			bReadDecPointVehicle := FALSE;	// Done in M_StateMachineNode_ADS
			bReadDecPointVehicleBusy := TRUE;
			bReturn := TRUE;			
		ELSE
	// NEW!!!
			// NOTE: iReadIndex is MagneMotion vehicle No
			REPEAT
				iReadIndex := iReadIndex + 1;
				IF (M_CheckVehicleOwned(iReadIndex)) THEN
					// Vehicle is owned by this cell... Read data from Track Server for this vehicle
					IF (M_CheckVehicleEventRead(iReadIndex)) THEN
						// Vehicle data is selected to be read! (event-based reading)
						EXIT;
					END_IF
				ELSIF (M_CheckVehicleSurvail(iReadIndex)) THEN
					// Vehicle is survailed by this cell (read data continously!)... Read data from Track Server for this vehicle
					EXIT;
				ELSIF (iReadIndex <> nDecisionPointVehicleNo) THEN
					// Not owned or surveilled or being handled by decision point. Delete any previous read data
					IF (iReadIndex > 0 AND iReadIndex <= MM_MAX_NUMBER_OF_VEHICLE_ELEMENTS) THEN
						aReadVehicleData[iReadIndex].stVehicle.bDataValid := FALSE;
					END_IF
				END_IF
				UNTIL (iReadIndex >= MM_MAX_NUMBER_OF_VEHICLE_ELEMENTS)
			END_REPEAT
			
			IF (iReadIndex <= MM_MAX_NUMBER_OF_VEHICLE_ELEMENTS) THEN
				// Build remote symbol name
				sPrefix := CONCAT(sObjectIDentifier, '.stTrackStatus');
				// Data pointer for received data
				pReadNodeData := ADR(aReadVehicleData[iReadIndex].stVehicle);
				// Header data size
				cbDataTotal := SIZEOF(aReadVehicleData[iReadIndex].stVehicle);
				
				// Specify nodes to read by variable name
				sTrackServerSymbol := CONCAT(sPrefix, '.aVehicles[');
				sTrackServerSymbol := CONCAT(sTrackServerSymbol, UINT_TO_STRING(iReadIndex));
				sTrackServerSymbol := CONCAT(sTrackServerSymbol, ']');
				
				// Remove this vehicle from the event-driven reading list
				M_VehicleToReadRemove(iReadIndex);
				
				bReturn := TRUE;
			ELSE
				// Read next type
				iReadIndex := 0;
				eReadType := E_OPC_NodeType.Paths;
				bReturn := FALSE;
			END_IF
	// NEW END!!!	
			// Select vehicle to read data from (only the vehicles this cell is responsible for)
(*			REPEAT
				iReadIndex := iReadIndex+1;
				IF (iReadIndex > MM_MAX_NUMBER_OF_VEHICLE_ELEMENTS) THEN
					EXIT;
				END_IF
				UNTIL (aReadCellData.stCell.anVehicles[iReadIndex] > 0)
			END_REPEAT
			IF (iReadIndex <= MM_MAX_NUMBER_OF_VEHICLE_ELEMENTS) THEN
				// Build remote symbol name
				sPrefix := CONCAT(sObjectIDentifier, '.stTrackStatus');
				// Data pointer for received data
				pReadNodeData := ADR(aReadVehicleData[aReadCellData.stCell.anVehicles[iReadIndex]].stVehicle);
				// Header data size
				cbDataTotal := SIZEOF(aReadVehicleData[aReadCellData.stCell.anVehicles[iReadIndex]].stVehicle);
				
				// Specify nodes to read by variable name
				sTrackServerSymbol := CONCAT(sPrefix, '.aVehicles[');
				sTrackServerSymbol := CONCAT(sTrackServerSymbol, UINT_TO_STRING(aReadCellData.stCell.anVehicles[iReadIndex]));
				sTrackServerSymbol := CONCAT(sTrackServerSymbol, ']');
				bReturn := TRUE;
			ELSE
				// Read next type
				iReadIndex := 0;
				eReadType := E_OPC_NodeType.Paths;
				bReturn := FALSE;
			END_IF		*)
		END_IF
		
	E_OPC_NodeType.Paths:
		// Select path to read data from
		REPEAT
			iReadIndex := iReadIndex+1;
			IF (iReadIndex > MM_MAX_NUMBER_OF_PATH_ELEMENTS) THEN
				EXIT;
			END_IF
			UNTIL (abControlledPaths[iReadIndex])
		END_REPEAT
		IF ((iReadIndex <= MM_MAX_NUMBER_OF_PATH_ELEMENTS) AND NOT tonSkipPathRead.Q) THEN	// Skip path reading when paths are started!
			// Build remote symbol name
			sPrefix := CONCAT(sObjectIDentifier, '.stTrackStatus');
			// Data pointer for received data
			pReadNodeData := ADR(aReadPathData[iReadIndex].stPathData);
			// Header data size
			cbDataTotal := SIZEOF(aReadPathData[iReadIndex].stPathData);
			
			// Specify nodes to read by variable name
			sTrackServerSymbol := CONCAT(sPrefix, '.aPaths[');
			sTrackServerSymbol := CONCAT(sTrackServerSymbol, UINT_TO_STRING(iReadIndex));
			sTrackServerSymbol := CONCAT(sTrackServerSymbol, ']');
			bReturn := TRUE;
		ELSE
			// Read next type
			iReadIndex := 0;
			eReadType := E_OPC_NodeType.Stations;
			bReturn := FALSE;
		END_IF
		
	E_OPC_NodeType.Stations:
		// Select Station to read data from
// TEST
		IF (M_CheckStationsRead()) THEN
			// Index for station data from track server has been found... Only read these stations
			REPEAT
				iReadIndex := iReadIndex+1;
				IF (iReadIndex > MM_MAX_NUMBER_OF_STATION_ELEMENTS) THEN
					EXIT;
				END_IF
				UNTIL (M_CheckStationIndex(iReadIndex))
			END_REPEAT
		ELSE
			// Index for station data from track server has NOT been found... Read data from all stations
			iReadIndex := iReadIndex + 1;
		END_IF
// TEST END
//		iReadIndex := iReadIndex+1;
		IF (iReadIndex <= MM_MAX_NUMBER_OF_STATION_ELEMENTS) THEN
			// Build remote symbol name
			sPrefix := CONCAT(sObjectIDentifier, '.stTrackStatus');
			// Data pointer
			pReadNodeData := ADR(aReadStationData[iReadIndex].stStationData);
			// Header data
			cbDataTotal := SIZEOF(aReadStationData[iReadIndex].stStationData);
			
			// Specify nodes to read by variable name
			sTrackServerSymbol := CONCAT(sPrefix, '.aStations[');
			sTrackServerSymbol := CONCAT(sTrackServerSymbol, UINT_TO_STRING(iReadIndex));
			sTrackServerSymbol := CONCAT(sTrackServerSymbol, ']');
			bReturn := TRUE;
		ELSE
			// Read next type
			iReadIndex := 0;
			eReadType := E_OPC_NodeType.Cells;
			bReturn := FALSE;
		END_IF
	
	E_OPC_NodeType.Cells:
		// Select Station to read data from
		iReadIndex := iThisCellIndex;
		IF (iReadIndex > 0 AND iReadIndex <= MM_MAX_NUMBER_OF_CELL_ELEMENTS) THEN
			// Build remote symbol name
			sPrefix := CONCAT(sObjectIDentifier, '.stTrackStatus');
			// Data pointer
			pReadNodeData := ADR(aReadCellData.stCell);
			// Header data
			cbDataTotal := SIZEOF(aReadCellData.stCell);
			
			// Specify nodes to read by variable name
			sTrackServerSymbol := CONCAT(sPrefix, '.aCells[');
			sTrackServerSymbol := CONCAT(sTrackServerSymbol, UINT_TO_STRING(iReadIndex));
			sTrackServerSymbol := CONCAT(sTrackServerSymbol, ']');
			bReturn := TRUE;

			// continue to next type after this read!
			iReadIndex := 0;
			bReadDecPointVehicle := TRUE;	// Force reading of the vehicle at decision point before other vehicles
			IF (NOT bReadDecPointCellDone) THEN
				bReadDecPointCell := TRUE;
			END_IF
			eReadType := E_OPC_NodeType.Vehicles;
		ELSE
			// Read next type
			iReadIndex := 0;
			bReadDecPointVehicle := TRUE;	// Force reading of the vehicle at decision point before other vehicles
			eReadType := E_OPC_NodeType.Vehicles;
			bReturn := FALSE;
		END_IF

END_CASE

M_InitNodeData_ADS := bReturn;
END_METHOD

METHOD PROTECTED M_InitNodeData_OPCUA : BOOL
VAR
	i		: UINT;
	sPrefix : STRING;
END_VAR
VAR
	cbDataTotal2 : UINT;
END_VAR
// NOTE!!!
// Maximum of 10 elements to read for each Node List reading!


(* Node data, init to use string identifier and set namespace index *)
FOR i:=1 TO nMaxNodeIDsInList BY 1 DO
	aNodeIDs[i].eIdentifierType := eUAIdentifierType_String;
	aNodeIDs[i].nNamespaceIndex := nNameSpaceIndexNodes;
END_FOR

nNoOfNodes := 0;
cbDataTotal := 0;

// TEST
eReadType := E_OPC_NodeType.Nodes;
iReadIndex := 1;

// Comm type selection
CASE eReadType OF
	E_OPC_NodeType.Vehicles:
		// Limit number of elements
		iReadIndex := LIMIT(1, iReadIndex, MM_MAX_NUMBER_OF_VEHICLE_ELEMENTS);
		// Build remote symbol name
		sPrefix := CONCAT(sObjectIDentifier, '.stTrackStatus.aVehicles[');
		sPrefix := CONCAT(sPrefix, UINT_TO_STRING(iReadIndex));
		sPrefix := CONCAT(sPrefix, ']');
		// Data pointer
		pReadNodeData := ADR(aReadVehicleData[iReadIndex]);
		// Header data
		cbDataTotal := SIZEOF(aReadVehicleData[iReadIndex].stReadListReturnInfo);
		
		// Specify nodes to read by variable name
		nNoOfNodes := nNoOfNodes + 1;
		aNodeIDs[nNoOfNodes].sIdentifier := CONCAT(sPrefix, '.nVehicleID');
		acbDatas[nNoOfNodes] := SIZEOF(aReadVehicleData[iReadIndex].nVehicleID);
		cbDataTotal := cbDataTotal + acbDatas[nNoOfNodes];
		
		nNoOfNodes := nNoOfNodes + 1;
		aNodeIDs[nNoOfNodes].sIdentifier := CONCAT(sPrefix, '.bVehiclePresent');
		acbDatas[nNoOfNodes] := SIZEOF(aReadVehicleData[iReadIndex].bVehiclePresent);
		cbDataTotal := cbDataTotal + acbDatas[nNoOfNodes];
		
		nNoOfNodes := nNoOfNodes + 1;
		aNodeIDs[nNoOfNodes].sIdentifier := CONCAT(sPrefix, '.nState');
		acbDatas[nNoOfNodes] := SIZEOF(aReadVehicleData[iReadIndex].nState);
		cbDataTotal := cbDataTotal + acbDatas[nNoOfNodes];
		
		nNoOfNodes := nNoOfNodes + 1;
		aNodeIDs[nNoOfNodes].sIdentifier := CONCAT(sPrefix, '.nPathID');
		acbDatas[nNoOfNodes] := SIZEOF(aReadVehicleData[iReadIndex].nPathID);
		cbDataTotal := cbDataTotal + acbDatas[nNoOfNodes];
		
		nNoOfNodes := nNoOfNodes + 1;
		aNodeIDs[nNoOfNodes].sIdentifier := CONCAT(sPrefix, '.fPosition');
		acbDatas[nNoOfNodes] := SIZEOF(aReadVehicleData[iReadIndex].fPosition);
		cbDataTotal := cbDataTotal + acbDatas[nNoOfNodes];
		
		nNoOfNodes := nNoOfNodes + 1;
		aNodeIDs[nNoOfNodes].sIdentifier := CONCAT(sPrefix, '.nTargetPathID');
		acbDatas[nNoOfNodes] := SIZEOF(aReadVehicleData[iReadIndex].nTargetPathID);
		cbDataTotal := cbDataTotal + acbDatas[nNoOfNodes];
		
		nNoOfNodes := nNoOfNodes + 1;
		aNodeIDs[nNoOfNodes].sIdentifier := CONCAT(sPrefix, '.fTargetPosition');
		acbDatas[nNoOfNodes] := SIZEOF(aReadVehicleData[iReadIndex].fTargetPosition);
		cbDataTotal := cbDataTotal + acbDatas[nNoOfNodes];
		
		nNoOfNodes := nNoOfNodes + 1;
		aNodeIDs[nNoOfNodes].sIdentifier := CONCAT(sPrefix, '.fVelocity');
		acbDatas[nNoOfNodes] := SIZEOF(aReadVehicleData[iReadIndex].fVelocity);
		cbDataTotal := cbDataTotal + acbDatas[nNoOfNodes];
				
		// Read next vehicle value
		iReadIndex := iReadIndex+1;;
		IF (iReadIndex > MM_MAX_NUMBER_OF_VEHICLE_ELEMENTS) THEN
			// Read next type
			iReadIndex := 0;
			eReadType := E_OPC_NodeType.Paths;
		END_IF

	E_OPC_NodeType.Paths:
		// Limit number of elements
		iReadIndex := LIMIT(1, iReadIndex, MM_MAX_NUMBER_OF_PATH_ELEMENTS);
		// Build remote symbol name
		sPrefix := CONCAT(sObjectIDentifier, '.stTrackStatus.aPaths[');
		sPrefix := CONCAT(sPrefix, UINT_TO_STRING(iReadIndex));
		sPrefix := CONCAT(sPrefix, ']');
		// Data pointer
		pReadNodeData := ADR(aReadPathData[iReadIndex]);
		
		// Header data
		cbDataTotal := SIZEOF(aReadPathData[iReadIndex].stReadListReturnInfo);
		
		// Specify nodes to read by variable name
		nNoOfNodes := nNoOfNodes + 1;
		aNodeIDs[nNoOfNodes].sIdentifier := CONCAT(sPrefix, '.nPathID');
		acbDatas[nNoOfNodes] := SIZEOF(aReadPathData[iReadIndex].nPathID);
		cbDataTotal := cbDataTotal + acbDatas[nNoOfNodes];

		nNoOfNodes := nNoOfNodes + 1;
		aNodeIDs[nNoOfNodes].sIdentifier := CONCAT(sPrefix, '.sCellID');
		acbDatas[nNoOfNodes] := SIZEOF(aReadPathData[iReadIndex].sCellID);
		cbDataTotal := cbDataTotal + acbDatas[nNoOfNodes];

		nNoOfNodes := nNoOfNodes + 1;
		aNodeIDs[nNoOfNodes].sIdentifier := CONCAT(sPrefix, '.bPathPresent');
		acbDatas[nNoOfNodes] := SIZEOF(aReadPathData[iReadIndex].bPathPresent);
		cbDataTotal := cbDataTotal + acbDatas[nNoOfNodes];

		nNoOfNodes := nNoOfNodes + 1;
		aNodeIDs[nNoOfNodes].sIdentifier := CONCAT(sPrefix, '.nState');
		acbDatas[nNoOfNodes] := SIZEOF(aReadPathData[iReadIndex].nState);
		cbDataTotal := cbDataTotal + acbDatas[nNoOfNodes];

		// Read next path value
		iReadIndex := iReadIndex+1;
		IF (iReadIndex > MM_MAX_NUMBER_OF_PATH_ELEMENTS) THEN
			// Read next type
			iReadIndex := 0;
			eReadType := E_OPC_NodeType.Nodes;
			//eReadType := E_OPC_NodeType.Vehicles;
		END_IF
		
		
	E_OPC_NodeType.Nodes:
		// Limit number of elements
		iReadIndex := LIMIT(1, iReadIndex, 10);
		// Build remote symbol name
		sPrefix := CONCAT(sObjectIDentifier, '.stTrackStatus');
		// Data pointer
		pReadNodeData := ADR(aReadNodeData[iReadIndex]);
		
		// Header data
		cbDataTotal := SIZEOF(aReadNodeData[iReadIndex].stReadListReturnInfo);
		cbDataTotal2 := SIZEOF(aReadNodeData[iReadIndex]);
		
		// Specify nodes to read by variable name
		nNoOfNodes := nNoOfNodes + 1;
		aNodeIDs[nNoOfNodes].sIdentifier := CONCAT(sPrefix, '.aNodes[');
		aNodeIDs[nNoOfNodes].sIdentifier := CONCAT(aNodeIDs[nNoOfNodes].sIdentifier, UINT_TO_STRING(iReadIndex));
		aNodeIDs[nNoOfNodes].sIdentifier := CONCAT(aNodeIDs[nNoOfNodes].sIdentifier, ']');
		acbDatas[nNoOfNodes] := SIZEOF(aReadNodeData[iReadIndex].stNodeData);
		cbDataTotal := cbDataTotal + acbDatas[nNoOfNodes];

		// Read next node value
		iReadIndex := iReadIndex+1;
		IF (iReadIndex > 10) THEN
			// Read next type
			iReadIndex := 0;
			eReadType := E_OPC_NodeType.Vehicles;
		END_IF

END_CASE
END_METHOD

METHOD PROTECTED M_MappingData
VAR_INPUT
END_VAR
VAR
	i			: USINT;
	iRes		: UINT;
END_VAR
// Handle the mapping data from OPC UA (stCommand)

CASE eMappingDataState OF
	// Init state
	E_MappingDataState.Undefined:
		eMappingDataState := E_MappingDataState.CheckRequest;
	
	// Check command data request
	E_MappingDataState.CheckRequest:
		IF ((stMappingIn.ChangeRequest <> stMappingOut.ChangeStatus) AND (stMappingIn.ChangeRequest > 0)) THEN
			// Check if changes is allowed on mapping data (from LC)
			IF (stAdditionalDataIn.MESHandShakes.DataChangeStatusTransportMapping = stMappingOut.DataChange) THEN
				stMappingOut.ChangeAcknowlegde := stMappingIn.ChangeRequest;
				stMappingOut.DataChange := stMappingOut.DataChange + 1;
				
				// Find vehicle ID with specified carrier ID
				iMappingDataVehicleID := M_CarrierIDToVehicleID(stMappingIn.Carrier.CarrierID);
	
				// Check vehicle number
				IF (iMappingDataVehicleID > 0) THEN
					eMappingDataState := E_MappingDataState.UpdateMappingData;
				ELSE
					eMappingDataState := E_MappingDataState.Error;
				END_IF
			END_IF	
		END_IF	
	
	// Perform data update
	E_MappingDataState.UpdateMappingData:
		iRes := M_CallUpdateVehicleMappingData(	nVehicleID := iMappingDataVehicleID,
												sCarrierID := stMappingIn.Carrier.CarrierID, 
												bTool := stMappingIn.Carrier.Tool, 
												sToolID := stMappingIn.Carrier.ToolID, 
												bMaterial := stMappingIn.Carrier.Material,
												sMaterialID := stMappingIn.Carrier.MaterialID 	);
		IF (iRes = 2) THEN
			// Success.
			eMappingDataState := E_MappingDataState.UpdateReworkData;
		ELSIF (iRes = 3) THEN
			// Error!
			eMappingDataState := E_MappingDataState.Error;
		END_IF
	
	// Perform rework update
	E_MappingDataState.UpdateReworkData:
		iRes := M_CallUpdateVehicleReworkData(	nVehicleID := iMappingDataVehicleID,
												sCarrierID := stMappingIn.Carrier.CarrierID,
												bNOK := stMappingIn.Carrier.NOK	); 
		IF (iRes = 2) THEN
			// Success..
			eMappingDataState := E_MappingDataState.Done;
		ELSIF (iRes = 3) THEN
			// Error!
			eMappingDataState := E_MappingDataState.Error;
		END_IF
	
	E_MappingDataState.Done:
		// Completed... Update output mapping data
		stMappingOut.ValidRequest := TRUE;
		stMappingOut.Carrier := stMappingIn.Carrier;
		stMappingOut.StationBuffer := stMappingIn.StationBuffer;
		stMappingOut.ChangeStatus := stMappingIn.ChangeRequest;
		stMappingOut.DataChange := stMappingOut.DataChange + 1;
		eMappingDataState := E_MappingDataState.Undefined;
	
	E_MappingDataState.Error:
		// Error... Valid request = FALSE
		stMappingOut.ValidRequest := FALSE;
		stMappingOut.ChangeStatus := stMappingIn.ChangeRequest;
		stMappingOut.DataChange := stMappingOut.DataChange + 1;
		eMappingDataState := E_MappingDataState.Undefined;
	
END_CASE
END_METHOD

METHOD PROTECTED M_ReworkData
VAR_INPUT
END_VAR
VAR
	i			: USINT;
	iRes		: UINT;
END_VAR
// Handle the mapping data from OPC UA (stCommand)

CASE eReworkDataState OF
	// Init state
	E_ReworkDataState.Undefined:
		bReworkValue := FALSE;
		iReworkDataStation := 0;
		iReworkDataStationNo := 0;
		eReworkDataState := E_ReworkDataState.CheckRequest;
	
	// Check command data request
	E_ReworkDataState.CheckRequest:
		FOR i := 1 TO 5 BY 1 DO
			/////////////////////////////////////////////////////////////////////////////////////////////////////////////////////
			// Rework completed from station (shoe rework is done handled)
			/////////////////////////////////////////////////////////////////////////////////////////////////////////////////////
			IF (abStation1ReworkDone[i]) THEN
				iReworkDataStation := i;
				iReworkDataStationNo := 1;

				// Check vehicle at station
				iReworkDataVehicleID := aStations[iReworkDataStation].stStationData1.nCurrentVehicleID;
				IF ((iReworkDataVehicleID > 0) AND (iReworkDataVehicleID <= MM_MAX_NUMBER_OF_VEHICLE_ELEMENTS) ) THEN
					// There is a vehicle on that station! Get the Carrier ID
					sReworkDataCarrierID := aReadVehicleData[iReworkDataVehicleID].stVehicle.sCarrierID;
					
					// Check carrier ID of vehicle
					IF (sReworkDataCarrierID <> '') THEN
						bReworkValue := FALSE;	// Set carrier status to rework NOT needed!
						eReworkDataState := E_ReworkDataState.UpdateReworkData;
					ELSE
						// Error!
						eReworkDataState := E_ReworkDataState.Error;
					
					END_IF
				ELSE
					// Error!
					eReworkDataState := E_ReworkDataState.Error;
				
				END_IF

				EXIT;
				
			ELSIF (abStation2ReworkDone[i]) THEN
				iReworkDataStation := i;
				iReworkDataStationNo := 2;

				iReworkDataVehicleID := aStations[iReworkDataStation].stStationData2.nCurrentVehicleID;
				IF ((iReworkDataVehicleID > 0) AND (iReworkDataVehicleID <= MM_MAX_NUMBER_OF_VEHICLE_ELEMENTS) ) THEN
					// There is a vehicle on that station! Get the Carrier ID
					sReworkDataCarrierID := aReadVehicleData[iReworkDataVehicleID].stVehicle.sCarrierID;
					
					// Check carrier ID of vehicle
					IF (sReworkDataCarrierID <> '') THEN
						bReworkValue := FALSE;	// Set carrier status to rework NOT needed!
						eReworkDataState := E_ReworkDataState.UpdateReworkData;
					ELSE
						// Error!
						eReworkDataState := E_ReworkDataState.Error;
					
					END_IF				
				ELSE
					// Error!
					eReworkDataState := E_ReworkDataState.Error;
				
				END_IF

				EXIT;

			/////////////////////////////////////////////////////////////////////////////////////////////////////////////////////
			// Rework request from station (shoe needs to be reworked)
			/////////////////////////////////////////////////////////////////////////////////////////////////////////////////////
			ELSIF (abStation1ReworkReq[i]) THEN
				iReworkDataStation := i;
				iReworkDataStationNo := 1;

				// Check vehicle at station
				iReworkDataVehicleID := aStations[iReworkDataStation].stStationData1.nCurrentVehicleID;
				IF ((iReworkDataVehicleID > 0) AND (iReworkDataVehicleID <= MM_MAX_NUMBER_OF_VEHICLE_ELEMENTS) ) THEN
					// There is a vehicle on that station! Get the Carrier ID
					sReworkDataCarrierID := aReadVehicleData[iReworkDataVehicleID].stVehicle.sCarrierID;
					
					// Check carrier ID of vehicle
					IF (sReworkDataCarrierID <> '') THEN
						bReworkValue := TRUE;	// Set carrier status to rework needed!
						eReworkDataState := E_ReworkDataState.UpdateReworkData;
					ELSE
						// Error!
						eReworkDataState := E_ReworkDataState.Error;
					
					END_IF
				ELSE
					// Error!
					eReworkDataState := E_ReworkDataState.Error;
				
				END_IF

				EXIT;
				
			ELSIF (abStation2ReworkReq[i]) THEN
				iReworkDataStation := i;
				iReworkDataStationNo := 2;

				iReworkDataVehicleID := aStations[iReworkDataStation].stStationData2.nCurrentVehicleID;
				IF ((iReworkDataVehicleID > 0) AND (iReworkDataVehicleID <= MM_MAX_NUMBER_OF_VEHICLE_ELEMENTS) ) THEN
					// There is a vehicle on that station! Get the Carrier ID
					sReworkDataCarrierID := aReadVehicleData[iReworkDataVehicleID].stVehicle.sCarrierID;
					
					// Check carrier ID of vehicle
					IF (sReworkDataCarrierID <> '') THEN
						bReworkValue := TRUE;	// Set carrier status to rework needed!
						eReworkDataState := E_ReworkDataState.UpdateReworkData;
					ELSE
						// Error!
						eReworkDataState := E_ReworkDataState.Error;
					
					END_IF				
				ELSE
					// Error!
					eReworkDataState := E_ReworkDataState.Error;
				
				END_IF

				EXIT;
			END_IF
		END_FOR
	
	// Perform rework update
	E_ReworkDataState.UpdateReworkData:
		iRes := M_CallUpdateVehicleReworkData(	nVehicleID := iReworkDataVehicleID,
												sCarrierID := sReworkDataCarrierID,
												bNOK := bReworkValue 	);
		IF (iRes = 2) THEN
			// Success..
			F_LogLine(CONCAT('TC_RWK: Vehicle ', CONCAT(UINT_TO_STRING(iReworkDataVehicleID), ' NOK set to %d')), BOOL_TO_DINT(bReworkValue));
			eReworkDataState := E_ReworkDataState.Done;
		ELSIF (iRes = 3) THEN
			// Error!
			eReworkDataState := E_ReworkDataState.Error;
		END_IF
	
	E_ReworkDataState.Done:
		// Completed... Wait until activation bit is sert to FALSE (when vehicle has been removed from station)
		IF (bReworkValue) THEN
			IF (iReworkDataStationNo = 1) THEN
				IF (NOT abStation1ReworkReq[iReworkDataStation]) THEN
					eReworkDataState := E_ReworkDataState.Undefined;		
				END_IF
	
			ELSIF (iReworkDataStationNo = 2) THEN
				IF (NOT abStation2ReworkReq[iReworkDataStation]) THEN
					eReworkDataState := E_ReworkDataState.Undefined;
				END_IF
	
			END_IF
		ELSE
			IF (iReworkDataStationNo = 1) THEN
				IF (NOT abStation1ReworkDone[iReworkDataStation]) THEN
					eReworkDataState := E_ReworkDataState.Undefined;		
				END_IF
	
			ELSIF (iReworkDataStationNo = 2) THEN
				IF (NOT abStation2ReworkDone[iReworkDataStation]) THEN
					eReworkDataState := E_ReworkDataState.Undefined;
				END_IF
	
			END_IF
		END_IF
	
	E_ReworkDataState.Error:
		// Error... Wait until activation bit is sert to FALSE (when vehicle has been removed from station)
		// TODO!!! Alarm!
		IF (bReworkValue) THEN
			IF (iReworkDataStationNo = 1) THEN
				IF (NOT abStation1ReworkReq[iReworkDataStation]) THEN
					eReworkDataState := E_ReworkDataState.Undefined;		
				END_IF
	
			ELSIF (iReworkDataStationNo = 2) THEN
				IF (NOT abStation2ReworkReq[iReworkDataStation]) THEN
					eReworkDataState := E_ReworkDataState.Undefined;
				END_IF
	
			END_IF
		ELSE
			IF (iReworkDataStationNo = 1) THEN
				IF (NOT abStation1ReworkDone[iReworkDataStation]) THEN
					eReworkDataState := E_ReworkDataState.Undefined;		
				END_IF
	
			ELSIF (iReworkDataStationNo = 2) THEN
				IF (NOT abStation2ReworkDone[iReworkDataStation]) THEN
					eReworkDataState := E_ReworkDataState.Undefined;
				END_IF
	
			END_IF
		END_IF

END_CASE
END_METHOD

METHOD PROTECTED M_Run : BOOL
VAR_INPUT
END_VAR
VAR
	i	: USINT;
END_VAR
// Get system time
fbGetTime(	NETID:= '',	// Local PLC 
			START:= NOT fbGetTime.START AND NOT fbGetTime.BUSY, 
			TMOUT:= T#5S	);

///////////////////////////////////////////////////////////////////////////////////////////////////////////////////
// FB's for method calling
///////////////////////////////////////////////////////////////////////////////////////////////////////////////////
	(* Handle server connect *)
	fbConnectMethod(	Execute				:= , 
						ServerUrl			:= sTrackServerUrl, 
						SessionConnectInfo	:= stConnectInfoMethod, 
						Timeout				:= T#10S, 
						ConnectionHdl		=> , 
						Done				=> , 
						Busy				=> , 
						Error				=> , 
						ErrorID				=> 	);
					
	(* Handle server dicconnect *)
	fbDisconnectMethod(	Execute				:= , 
						ConnectionHdl		:= nConnectHdlMethod, 
						Timeout				:= T#10S, 
						Done				=> , 
						Busy				=> , 
						Error				=> , 
						ErrorID				=> 	);
						
	(* Get namepsace *)
	fbGetNamespaceMethod(	Execute				:= , 
							ConnectionHdl		:= nConnectHdlMethod, 
							NamespaceUri		:= sNameSpaceUri, 
							Timeout				:= T#10S, 
							NamespaceIndex		=> , 
							Done				=> , 
							Busy				=> , 
							Error				=> , 
							ErrorID				=> 	);
	
	(* Get method handle *)
	stObjectNodeID.nNamespaceIndex := nNameSpaceIndexMethod;
	stObjectNodeID.sIdentifier := sObjectIDentifier;
	stMethodNodeID.nNamespaceIndex := nNameSpaceIndexMethod;
	stMethodNodeID.sIdentifier := sMethodIdentifier;
	fbGetHandleMethod(	Execute				:= , 
						ConnectionHdl		:= nConnectHdlMethod, 
						ObjectNodeID		:= stObjectNodeID, 
						MethodNodeID		:= stMethodNodeID, 
						Timeout				:= T#10S, 
						MethodHdl			=> , 
						Done				=> , 
						Busy				=> , 
						Error				=> , 
						ErrorID				=>	);
	
	(* Call method *)
	fbCallMethod(	Execute					:= , 
					ConnectionHdl			:= nConnectHdlMethod, 
					MethodHdl				:= nHandleMethod, 
					nNumberOfInputArguments	:= , 
					pInputArgInfo			:= , 
					cbInputArgInfo			:= , 
					pInputArgData			:= , 
					cbInputArgData			:= , 
					pInputWriteData			:= 0,
					cbInputWriteData		:= 0,
					nNumberOfOutputArguments:= , 
					pOutputArgInfo			:= , 
					cbOutputArgInfo			:= , 
					pOutputArgInfoAndData	:= , 
					cbOutputArgInfoAndData	:= , 
					Timeout					:= T#10S, 
					cbRead_R				=> , 
					Done					=> , 
					Busy					=> , 
					Error					=> , 
					ErrorID					=> );
	
	(* Release method handle *)
	fbReleaseHandleMethod(	Execute			:= , 
							ConnectionHdl	:= nConnectHdlMethod, 
							MethodHdl		:= nHandleMethod, 
							Timeout			:= T#10S, 
							Done			=> , 
							Busy			=> , 
							Error			=> , 
							ErrorID			=> 	);

///////////////////////////////////////////////////////////////////////////////////////////////////////////////////
// FB's for method calling
///////////////////////////////////////////////////////////////////////////////////////////////////////////////////
	(* Handle server connect *)
	fbConnectNodes(	Execute				:= , 
					ServerUrl			:= sTrackServerUrl, 
					SessionConnectInfo	:= stConnectInfoNodes, 
					Timeout				:= T#10S, 
					ConnectionHdl		=> , 
					Done				=> , 
					Busy				=> , 
					Error				=> , 
					ErrorID				=> 	);
					
	(* Handle server dicconnect *)
	fbDisconnectNodes(	Execute				:= , 
						ConnectionHdl		:= nConnectHandleNodes, 
						Timeout				:= T#10S, 
						Done				=> , 
						Busy				=> , 
						Error				=> , 
						ErrorID				=> 	);
						
	(* Get namepsace *)
	fbGetNamespaceNodes(	Execute				:= , 
						ConnectionHdl		:= nConnectHandleNodes, 
						NamespaceUri		:= sNameSpaceUri, 
						Timeout				:= T#10S, 
						NamespaceIndex		=> , 
						Done				=> , 
						Busy				=> , 
						Error				=> , 
						ErrorID				=> 	);
	
	(* Get node handle *)
	fbGetHandleNodes(	Execute				:= , 
						ConnectionHdl		:= nConnectHandleNodes, 
						NodeIDCount			:= nNoOfNodes,
						NodeIDs				:= aNodeIDs, 
						Timeout				:= T#10S, 
						NodeHdls			=> , 
						Done				=> , 
						Busy				=> , 
						Error				=> , 
						ErrorID				=> 	);
		
	(* Read node data *)
	fbReadNodes(	Execute:= , 
					ConnectionHdl			:= nConnectHandleNodes,
					NodeHdlCount			:= nNoOfNodes,
					NodeHdls				:= anHandleNodes, 
					stNodeAddInfo			:= astNodeAddInfo, 
					pVariable				:= pReadNodeData, 
					cbData					:= acbDatas,
					cbDataTotal				:= cbDataTotal, 
					Timeout					:= T#10S, 
					Done					=> , 
					Busy					=> , 
					Error					=> , 
					ErrorID					=> , 
					cbData_R				=> 	);
					
	(* Release node handle list *)
	fbReleaseHandleNodes(	Execute			:= , 
							ConnectionHdl	:= nConnectHandleNodes, 
							NodeHdlCount	:= nNoOfNodes, 
							NodeHdls		:= anHandleNodes, 
							Timeout			:= T#10S, 
							NodeErrorIDs	=> , 
							Done			=> , 
							Busy			=> , 
							Error			=> , 
							ErrorID			=> 	);
	
	(* Read interval *)
	tonReadInterval(	IN	:= ,
						PT	:= REAL_TO_TIME(rReadInterval * 1000.0),
						Q	=> ,
						ET	=> 	);
						
	(* Error automatic reset delay *)
	tonErrorReset(		IN	:= ,
						PT	:= REAL_TO_TIME(rErrorResetDelay * 1000.0),
						Q	=> ,
						ET	=> 	);

// Update Additional Data variables
	stAdditionaldataOut.bConnectedMethod := bConnectedMethod;
	stAdditionaldataOut.bConnectedNode := bConnectedNode;
	stAdditionaldataOut.bTrackReady := P_bTrackReady;
END_METHOD

METHOD PROTECTED M_StateMachine : BOOL
VAR_INPUT
END_VAR
VAR
	iRes	: INT;
	i		: UINT;
END_VAR

CASE eTrackState OF
	E_TrackState.Undefined:
		bStarted := FALSE;
		bSuspended := FALSE;
		iStationID := 1;
		iPathID := 1;
		iPathIndex := 1;
		IF (bConnectedMethod AND bConnectedNode) THEN
			// Communication connections established
			IF (bEnable) THEN
				eTrackState := E_TrackState.CheckInitDone;
			END_IF
		END_IF
	
	E_TrackState.CheckInitDone:
		// Check if track has been setup from this cell already on the track server
		iRes := M_CallGetCellIndex(sCellID);
		IF (iRes = 2) THEN
			// Success... Init done
			// Save found index
			iThisCellIndex := stGetCellIndexData.stOutput.nCellIndex;
			IF (iThisCellIndex > 0) THEN
				bTrackInitDone := TRUE;
				eTrackState := E_TrackState.Starting;
			ELSE
				bTrackInitDone := FALSE;
				bStationData1Done := FALSE;
				bStationData2Done := FALSE;
				// Clear station index
				FOR i := 1 TO 5 BY 1 DO
					iThisStationIndex[i] := 0;
				END_FOR
				eTrackState := E_TrackState.WaitAllowInit;
			END_IF
		ELSIF (iRes = 3) THEN
			// Error!
			// Clear station index
			FOR i := 1 TO 5 BY 1 DO
				iThisStationIndex[i] := 0;
			END_FOR
			eTrackState := E_TrackState.WaitAllowInit;
		END_IF
	
//	E_TrackState.InitDecisionPoint:
//		// Initialized with stations
//		eTrackState := E_TrackState.InitStations;
	
	E_TrackState.WaitAllowInit:
		// Initialized with stations
		IF (stAdditionalDataIn.bAllowInit) THEN
			stAdditionalDataIn.bAllowInit := FALSE;
			eTrackState := E_TrackState.InitStations;
		ELSIF (NOT bEnable OR NOT bConnectedMethod OR NOT bConnectedNode) THEN
			eTrackState := E_TrackState.Undefined;
		END_IF

	E_TrackState.InitStations:
		IF (aStations[iStationID].bPresent) THEN
			IF (aStations[iStationID].stStationData2.stLocation.nPathID > 0) THEN
				// Double position station
				iRes := M_CallAddStationDouble(nStationNo := iStationID);
				IF (iRes = 2) THEN
					// Success... Next station
					iStationID := iStationID + 1;
				ELSIF (iRes = 3) THEN
					// Error!
					// TODO!!!
					;				
				END_IF
			ELSE
				// Single position station
				iRes := M_CallAddStationSingle(nStationNo := iStationID);
				IF (iRes = 2) THEN
					// Success... Next station
					iStationID := iStationID + 1;
				ELSIF (iRes = 3) THEN
					// Error!
					// TODO!!!
					;				
				END_IF
			END_IF
		ELSE
			// Not enabled... Next station
			iStationID := iStationID + 1;
		END_IF
		IF (iStationID >= 5) THEN
			// All added
			iStationID := 1;
//			eTrackState := E_TrackState.InitPathsStations;	// init paths from stations, traffic lights and decision point 
			eTrackState := E_TrackState.SetPreBufferAdjust;
		END_IF
		
	E_TrackState.SetPreBufferAdjust:
		IF (aStations[iStationID].bPresent) THEN
			IF (aStationPreBufAdj[iStationID] <> 0.0) THEN
				iRes := M_CallAdjustBufferPosition(	nStationNo := iStationID,
													eBufferType := E_MMStationBuffer.eMMStationBuffer_PreProcess,
													rDistance := aStationPreBufAdj[iStationID]	);
				IF (iRes = 2) THEN
					// Success... Next station
					iStationID := iStationID + 1;
				ELSIF (iRes = 3) THEN
					// Error!
					// TODO!!!
					;
				END_IF
				
			ELSE
				// No adustment needed
				iStationID := iStationID + 1;
			END_IF
		ELSE
			// Not enabled... Next station
			iStationID := iStationID + 1;
		END_IF
		IF (iStationID >= 5) THEN
			// All checked/adjusted
			iStationID := 1;
			eTrackState := E_TrackState.SetPostBufferAdjust;
		END_IF
		
	E_TrackState.SetPostBufferAdjust:
		IF (aStations[iStationID].bPresent) THEN
			IF (aStationPostBufAdj[iStationID] <> 0.0) THEN
				iRes := M_CallAdjustBufferPosition(	nStationNo := iStationID,
													eBufferType := E_MMStationBuffer.eMMStationBuffer_PostProcess,
													rDistance := aStationPostBufAdj[iStationID]	);
				IF (iRes = 2) THEN
					// Success... Next station
					iStationID := iStationID + 1;
				ELSIF (iRes = 3) THEN
					// Error!
					// TODO!!!
					;
				END_IF
				
			ELSE
				// No adustment needed
				iStationID := iStationID + 1;
			END_IF
		ELSE
			// Not enabled... Next station
			iStationID := iStationID + 1;
		END_IF
		IF (iStationID >= 5) THEN
			// All checked/adjusted
			iStationID := 1;
			eTrackState := E_TrackState.InitPaths;
		END_IF
		
	// Create/init paths on track server for this cell
	E_TrackState.InitPaths:	
		IF (aPaths[iPathID] > 0) THEN
			iRes := M_CallAddPath(nPathNo := aPaths[iPathID]);
			IF (iRes = 2) THEN
				// Success... Next Path
				abControlledPaths[aPaths[iPathID]] := TRUE;
				iPathID := iPathID + 1;
			ELSIF (iRes = 3) THEN
				// Error!
				// TODO!!!
				;
			END_IF
		ELSE
			// All added
			iPathID := 1;
			eTrackState := E_TrackState.InitGetCellIndex;
		END_IF
(*		
	// Create/init paths on track server for this cell
	E_TrackState.InitPathsStations:	
		IF (aStations[iStationID].bPresent) THEN
			IF (NOT bStationData1Done) THEN
				iRes := M_CallAddPath(nPathNo := aStations[iStationID].stStationData1.stLocation.nPathID);
				IF (iRes = 2) THEN
					// Success... Next station
					abControlledPaths[aStations[iStationID].stStationData1.stLocation.nPathID] := TRUE;
					bStationData1Done := TRUE;
					IF (aStations[iStationID].stStationData1.stLocation.nPathID = aStations[iStationID].stStationData2.stLocation.nPathID) THEN
						// Station 2 is on the same path
						bStationData2Done := TRUE;
						iStationID := iStationID + 1;						
					ELSE
						// Station 2 is on a different path
						
					END_IF
				ELSIF (iRes = 3) THEN
					// Error!
					// TODO!!!
					;
				END_IF
			ELSIF (NOT bStationData2Done) THEN
				iRes := M_CallAddPath(nPathNo := aStations[iStationID].stStationData2.stLocation.nPathID);
				IF (iRes = 2) THEN
					// Success... Next station
					abControlledPaths[aStations[iStationID].stStationData2.stLocation.nPathID] := TRUE;
					bStationData2Done := TRUE;
					iStationID := iStationID + 1;
				ELSIF (iRes = 3) THEN
					// Error!
					// TODO!!!
					;
				END_IF
			END_IF
		ELSE
			// Not enabled... Next station
			iStationID := iStationID + 1;
		END_IF
		IF (iStationID >= 5) THEN
			// All added
			iStationID := 1;
			eTrackState := E_TrackState.InitPathsDecisionPoint;
		END_IF
	
	// Create/init paths on track server for this cell
	E_TrackState.InitPathsDecisionPoint:	
		IF (aStations[iStationID].bPresent) THEN
			iRes := M_CallAddPath(nPathNo := aStations[iStationID].stDecisionLocation.nPathID);
			IF (iRes = 2) THEN
				// Success... Next station
				abControlledPaths[aStations[iStationID].stDecisionLocation.nPathID] := TRUE;
				iStationID := iStationID + 1;
			ELSIF (iRes = 3) THEN
				// Error!
				// TODO!!!
				;
			END_IF
		ELSE
			// Not enabled... Next station
			iStationID := iStationID + 1;
		END_IF
		IF (iStationID >= 5) THEN
			// All added
			iStationID := 1;
			eTrackState := E_TrackState.InitPathsTrafficLight;
		END_IF

	// Create/init paths on track server for this cell
	E_TrackState.InitPathsTrafficLight:	
		IF (stTrafficLightLocation.nPathID > 0) THEN
			iRes := M_CallAddPath(nPathNo := stTrafficLightLocation.nPathID);	
			IF (iRes = 2) THEN
				// Success
				abControlledPaths[stTrafficLightLocation.nPathID] := TRUE;
				eTrackState := E_TrackState.InitGetCellIndex;
			ELSIF (iRes = 3) THEN
				// Error!
				// TODO!!!
				;
			END_IF
		ELSE
			eTrackState := E_TrackState.InitGetCellIndex;			
		END_IF
*)
	E_TrackState.InitGetCellIndex:
		iRes := M_CallGetCellIndex(sCellID);
		IF (iRes = 2) THEN
			// Success... Init done
			// Save found index
			iThisCellIndex := stGetCellIndexData.stOutput.nCellIndex;
			bTrackInitDone := TRUE;
			eTrackState := E_TrackState.Resetting;
		ELSIF (iRes = 3) THEN
			// Error!
			// TODO!!!
			;
		END_IF	
	
	E_TrackState.Starting:
		IF (abControlledPaths[iPathID]) THEN
			// This path is controlled by this cell
			iRes := M_CallStartPath(nPathNo := iPathID);
			IF (iRes = 2) THEN
				// Success... Next station
				iPathID := iPathID + 1;
			ELSIF (iRes = 3) THEN
				// Error!
				// TODO!!!
				;
			END_IF
			
		ELSE
			iPathID := iPathID + 1;
		END_IF
		IF (iPathID >= MM_MAX_NUMBER_OF_PATH_ELEMENTS) THEN
			// All started
			iPathID := 1;
			bPathsOperational := TRUE;
			bPathsSuspended := FALSE;
			eTrackState := E_TrackState.StartCheck;
		END_IF
	
	E_TrackState.StartCheck:
		IF (abControlledPaths[iPathID]) THEN
			// Is this path controlled by this cell
			IF (aReadPathData[iPathID].stPathData.bPathPresent AND (aReadPathData[iPathID].stPathData.nState = E_MMPathState.eMMPathState_Operational)) THEN
				// This path is operational
				bPathsOperational := bPathsOperational AND TRUE;
			ELSE
				// Not operational
				bPathsOperational := FALSE;
			END_IF
			IF (aReadPathData[iPathID].stPathData.nMotionStatus = E_MMPathMotionStatus.eMMPathMotionStatus_SuspendedByCommand) THEN
				// This path is suspended!
				bPathsSuspended := TRUE;
			END_IF
		END_IF
		iPathID := iPathID + 1;
		IF (iPathID > MM_MAX_NUMBER_OF_PATH_ELEMENTS) THEN
			IF (bPathsOperational) THEN
				// All paths OK... Continue
				iPathID := 1;
				eTrackState := E_TrackState.InitTrafficLight;
			ELSIF (NOT bEnable) THEN
				// Stop
				eTrackState := E_TrackState.Undefined;			
			ELSE
				// All paths NOT OK!
				bPathsOperational := TRUE;
				bPathsSuspended := FALSE;
				iPathID := 1;
			END_IF
		END_IF
	
	E_TrackState.InitTrafficLight:
		// Check if Traffic light is defined!
		IF (stTrafficLightLocation.nPathID > 0) THEN
			iRes := M_CallAddTrafficLight(	nTrafficLightID := 1,
											nPathID := stTrafficLightLocation.nPathID,
											fPosition := stTrafficLightLocation.fPosition);
			IF (iRes = 2) THEN
				// Success... Init done
				eTrackState := E_TrackState.InitTrafficLight2;
			ELSIF (iRes = 3) THEN
				// Error!
				// TODO!!!
				;				
			END_IF
		ELSE
			eTrackState := E_TrackState.InitTrafficLight2;
		END_IF
	
	E_TrackState.InitTrafficLight2:
		// Check if Traffic light 2 is defined!
		IF (stTrafficLight2Location.nPathID > 0) THEN
			iRes := M_CallAddTrafficLight(	nTrafficLightID := 2,
											nPathID := stTrafficLight2Location.nPathID,
											fPosition := stTrafficLight2Location.fPosition);
			IF (iRes = 2) THEN
				// Success... Init done
				eTrackState := E_TrackState.InitPathSegment;
			ELSIF (iRes = 3) THEN
				// Error!
				// TODO!!!
				;				
			END_IF
		ELSE
			eTrackState := E_TrackState.InitPathSegment;
		END_IF

	E_TrackState.InitPathSegment:
		// Check if Path Segment is defined!
		IF (stExitPointSeg1LocBegin.nPathID > 0) THEN
			iRes := M_CallAddPathSegment(	iSegmentNo := 1,
											nPathNo := stExitPointSeg1LocBegin.nPathID,
											rBeginPosition := stExitPointSeg1LocBegin.fPosition,
											rEndPosition := stExitPointSeg1LocEnd.fPosition);
			IF (iRes = 2) THEN
				// Success... Init done
				eTrackState := E_TrackState.InitPathSegment2;
			ELSIF (iRes = 3) THEN
				// Error!
				// TODO!!!
				;				
			END_IF
		ELSE
			eTrackState := E_TrackState.InitPathSegment2;
		END_IF
	
	E_TrackState.InitPathSegment2:
		// Check if Path Segment is defined!
		IF (stExitPointSeg2LocBegin.nPathID > 0) THEN
			iRes := M_CallAddPathSegment(	iSegmentNo := 2,
											nPathNo := stExitPointSeg2LocBegin.nPathID,
											rBeginPosition := stExitPointSeg2LocBegin.fPosition,
											rEndPosition := stExitPointSeg2LocEnd.fPosition);
			IF (iRes = 2) THEN
				// Success... Init done
				eTrackState := E_TrackState.InitVehicles;
			ELSIF (iRes = 3) THEN
				// Error!
				// TODO!!!
				;				
			END_IF
		ELSE
			eTrackState := E_TrackState.InitVehicles;
		END_IF
	
	E_TrackState.InitVehicles:
		IF (bVehicleInitDone) THEN
			// Init done, go to started!
			eTrackState := E_TrackState.Started;
		ELSE
			iVehicleIndex := iVehicleIndex + 1;	// Start from 0!
			IF (aReadCellData.stCell.anVehicles[iVehicleIndex] > 0) THEN
				// Handle this vehicle
				iRes := M_CallMoveVehicleToScanner(	eInputType := E_MMVehicleInputType.eMMVehicleInputType_VehicleID,
													sInput := UINT_TO_STRING(aReadCellData.stCell.anVehicles[iVehicleIndex]),
													eDirection := E_MMDirection.eMMDirection_Forward, 
													fVelocity := 1,
													fAcceleration := 1 	);
				IF (iRes = 2) THEN
					// Next vehicle
					iVehicleIndex := iVehicleIndex + 1;
				ELSIF (iRes = 3) THEN
					// Error!
					// TODO!!!
					;
				END_IF
			ELSE
				// Next vehicle
				iVehicleIndex := iVehicleIndex + 1;
			END_IF
			IF (iVehicleIndex >= MM_MAX_NUMBER_OF_VEHICLE_ELEMENTS) THEN
				// All inited
				bVehicleInitDone := TRUE;
				iVehicleIndex := 0;
				eTrackState := E_TrackState.Started;
			END_IF
		END_IF
		
	E_TrackState.Started:
		bStarted := TRUE;
		IF (NOT bEnable) THEN
			// Disable
			eTrackState := E_TrackState.Undefined;
		ELSIF (iThisCellIndex <= 0) THEN
			// Re-Init cell index from track server
			iRes := M_CallGetCellIndex(sCellID);
			IF (iRes = 2) THEN
				// Success... Init done
				// Save found index
				iThisCellIndex := stGetCellIndexData.stOutput.nCellIndex;
			ELSIF (iRes = 3) THEN
				// Error!
				// TODO!!!
				;
			END_IF	
		ELSIF (bSuspend) THEN
			// Activate suspend on paths
			eTrackState := E_TrackState.Suspend;
		ELSIF (bPathsSuspended AND NOT bSuspend) THEN
			// Some paths are suspended and should not be
			eTrackState := E_TrackState.Resume;
		END_IF

	E_TrackState.Suspend:
		IF ( abControlledPaths[iPathID] AND (aReadPathData[iPathID].stPathData.nMotionStatus <> E_MMPathMotionStatus.eMMPathMotionStatus_SuspendedByCommand) ) THEN
			// This path is controlled by this cell and is not suspended
			iRes := M_CallSuspendPath(nPathNo := iPathID);
			IF (iRes = 2) THEN
				// Success... Next station
				iPathID := iPathID + 1;
			ELSIF (iRes = 3) THEN
				// Error!
				// TODO!!!
				;
			END_IF
		ELSE
			iPathID := iPathID + 1;
		END_IF
		IF (iPathID >= MM_MAX_NUMBER_OF_PATH_ELEMENTS) THEN
			// All suspended
			iPathID := 1;
			bPathsSuspended := TRUE;
			eTrackState := E_TrackState.Suspending;
		END_IF
		
	E_TrackState.Suspending:
		IF (abControlledPaths[iPathID]) THEN
			// Is this path controlled by this cell
			IF (aReadPathData[iPathID].stPathData.nMotionStatus = E_MMPathMotionStatus.eMMPathMotionStatus_SuspendedByCommand) THEN
				// This path is suspended
				bPathsSuspended := bPathsSuspended AND TRUE;
			ELSE
				// Not operational
				bPathsSuspended := FALSE;
			END_IF
		END_IF
		iPathID := iPathID + 1;
		IF (iPathID > MM_MAX_NUMBER_OF_PATH_ELEMENTS) THEN
			IF (bPathsSuspended) THEN
				// All paths Suspended... Continue
				iPathID := 1;
				eTrackState := E_TrackState.Suspended;
			ELSIF (NOT bEnable) THEN
				// Stop
				eTrackState := E_TrackState.Undefined;			
			ELSE
				// All paths NOT Suspended!
				iPathID := 1;
				bPathsSuspended := TRUE;
			END_IF
		END_IF		
	
	E_TrackState.Suspended:
		IF (NOT bSuspend) THEN
			bSuspended := FALSE;
			eTrackState := E_TrackState.Resume;
		ELSIF (NOT bEnable) THEN
			eTrackState := E_TrackState.Undefined;			
		END_IF
		
	E_TrackState.Resume:
		IF ( abControlledPaths[iPathID] AND aReadPathData[iPathID].stPathData.nMotionStatus = E_MMPathMotionStatus.eMMPathMotionStatus_SuspendedByCommand ) THEN
			// This path is controlled by this cell
			iRes := M_CallResumePath(nPathNo := iPathID);
			IF (iRes = 2) THEN
				// Success... Next station
				iPathID := iPathID + 1;
			ELSIF (iRes = 3) THEN
				// Error!
				// TODO!!!
				;
			END_IF
			
		ELSE
			iPathID := iPathID + 1;
		END_IF
		IF (iPathID >= MM_MAX_NUMBER_OF_PATH_ELEMENTS) THEN
			// All started
			iPathID := 1;
			bPathsResumed := TRUE;
			eTrackState := E_TrackState.Resuming;
		END_IF
	
	E_TrackState.Resuming:
		IF (abControlledPaths[iPathID]) THEN
			// Is this path controlled by this cell
			IF (aReadPathData[iPathID].stPathData.nMotionStatus <> E_MMPathMotionStatus.eMMPathMotionStatus_SuspendedByCommand) THEN
				// This path is operational
				bPathsResumed := bPathsResumed AND TRUE;
			ELSE
				// Not operational
				bPathsResumed := FALSE;
			END_IF
		END_IF
		iPathID := iPathID + 1;
		IF (iPathID > MM_MAX_NUMBER_OF_PATH_ELEMENTS) THEN
			IF (bPathsResumed) THEN
				// All paths Resumed... Continue
				iPathID := 1;
				bPathsSuspended := FALSE;
				eTrackState := E_TrackState.Started;
			ELSIF (NOT bEnable) THEN
				// Stop
				eTrackState := E_TrackState.Undefined;			
			ELSE
				// All paths NOT OK!
				bPathsResumed := TRUE;
				iPathID := 1;
			END_IF
		END_IF		
	
	E_TrackState.Resetting:
		IF (abControlledPaths[iPathID]) THEN
			// This path is controlled by this cell
			iRes := M_CallResetPath(nPathNo := iPathID);
			IF (iRes = 2) THEN
				// Success... Next station
				iPathID := iPathID + 1;
			ELSIF (iRes = 3) THEN
				// Error!
				// TODO!!!
				;
			END_IF
			
		ELSE
			iPathID := iPathID + 1;
		END_IF
		IF (iPathID >= MM_MAX_NUMBER_OF_PATH_ELEMENTS) THEN
			// All reset
			iPathID := 1;
			eTrackState := E_TrackState.ResetWait;
		END_IF

	E_TrackState.ResetWait:
		tonResetTime(IN := TRUE, PT := T#4S);
		IF (tonResetTime.Q) THEN
			tonResetTime(IN := FALSE);
			eTrackState := E_TrackState.ResetCheck;						
		END_IF
	
	E_TrackState.ResetCheck:
		IF (abControlledPaths[iPathID]) THEN
			// Is this path controlled by this cell
			IF (aReadPathData[iPathID].stPathData.bPathPresent AND
				( (aReadPathData[iPathID].stPathData.nState = E_MMPathState.eMMPathState_Operational) OR (aReadPathData[iPathID].stPathData.nState = E_MMPathState.eMMPathState_Initialization) )) THEN
				// This path is operational or reset completed
				bPathsReset := bPathsReset AND TRUE;
			ELSE
				// Not operational
				bPathsReset := FALSE;
			END_IF
		END_IF
		iPathID := iPathID + 1;
		IF (iPathID > MM_MAX_NUMBER_OF_PATH_ELEMENTS) THEN
			IF (bPathsReset) THEN
				// All paths OK... Continue
				iPathID := 1;
				eTrackState := E_TrackState.Idle;
			ELSIF (NOT bEnable) THEN
				// Stop
				eTrackState := E_TrackState.Undefined;			
			ELSE
				// All paths NOT OK!
				bPathsReset := TRUE;
				iPathID := 1;
			END_IF
		END_IF

	E_TrackState.Idle:
		IF (bEnable) THEN
			eTrackState := E_TrackState.Undefined;
		END_IF

	E_TrackState.Error:

END_CASE

tonSkipPathRead(IN := (eTrackState = E_TrackState.Started),
				PT := T#5S,
				Q => ,
				ET =>	);

// Shut down track from OPC-UA interface
IF (stAdditionalDataIn.bShutDown) THEN
	stAdditionalDataIn.bShutDown := FALSE;
	bEnable := FALSE;
END_IF
END_METHOD

METHOD PROTECTED M_StateMachineMethod : BOOL
VAR_INPUT
END_VAR
CASE eStateMethod OF
	E_TrackClientState.Disconnected:
		bConnectedMethod := FALSE;
		bBusyMethod := FALSE;
		fbConnectMethod.Execute := FALSE;
		fbDisconnectMethod.Execute := FALSE;
		fbGetNamespaceMethod.Execute := FALSE;
		fbGetHandleMethod.Execute := FALSE;
		fbCallMethod.Execute := FALSE;
		fbReleaseHandleMethod.Execute := FALSE;
		IF (bEnable) THEN
			bErrorMethod := FALSE;
			nErrorMethodID := 0;
			eStateMethod := E_TrackClientState.Connecting;
		END_IF
	
	E_TrackClientState.Connecting:
		IF (fbConnectMethod.Execute AND NOT fbConnectMethod.Busy) THEN
			fbConnectMethod.Execute := FALSE;
			IF (NOT fbConnectMethod.Error) THEN
				(* Connected *)
				nConnectHdlMethod := fbConnectMethod.ConnectionHdl;
				eStateMethod := E_TrackClientState.GetNamespaceIndex;
			ELSE
				(* Error during connection *)
				bErrorMethod := TRUE;
				nErrorMethodID := fbConnectMethod.ErrorID;
				eLastErrorMethodID := nErrorMethodID;
				nConnectHdlMethod := 0;
				eStateMethod := E_TrackClientState.Error;
			END_IF
		ELSE
			fbConnectMethod.Execute := TRUE;		
		END_IF
	
	E_TrackClientState.GetNamespaceIndex:
		IF (fbGetNamespaceMethod.Execute AND NOT fbGetNamespaceMethod.Busy) THEN
			fbGetNamespaceMethod.Execute := FALSE;
			IF (NOT fbGetNamespaceMethod.Error) THEN
				nNameSpaceIndexMethod := fbGetNamespaceMethod.NamespaceIndex;
				eStateMethod := E_TrackClientState.Connected;
			ELSE
				(* Error during get namepsace index *)
				nNameSpaceIndexMethod := 0;
				bErrorMethod := TRUE;
				nErrorMethodID := fbGetNamespaceMethod.ErrorID;
				eStateMethod := E_TrackClientState.Disconnecting;
			END_IF
		ELSE
			fbGetNamespaceMethod.Execute := TRUE;
		END_IF
	
	E_TrackClientState.Connected:
		bConnectedMethod := TRUE;
		bBusyMethod := FALSE;
		IF (NOT bEnable) THEN
			bConnectedMethod := FALSE;
			eStateMethod := E_TrackClientState.Disconnecting;
		ELSIF (bCallMethod) THEN
			bCallMethod := FALSE;
			bBusyMethod := TRUE;
			eStateMethod := E_TrackClientState.GetHandle;
		END_IF
		
	E_TrackClientState.GetHandle:
		IF (fbGetHandleMethod.Execute AND NOT fbGetHandleMethod.Busy) THEN
			fbGetHandleMethod.Execute := FALSE;
			IF (NOT fbGetHandleMethod.Error) THEN
				nHandleMethod := fbGetHandleMethod.MethodHdl;
				eStateMethod := E_TrackClientState.Execute;
			ELSE
				(* Error during get method handle *)
				nHandleMethod := 0;
				bErrorMethod := TRUE;
				nErrorMethodID := fbGetHandleMethod.ErrorID;
				eStateMethod := E_TrackClientState.Disconnecting;
			END_IF
		ELSE
			fbGetHandleMethod.Execute := TRUE;
		END_IF

	E_TrackClientState.Execute:
		IF (fbCallMethod.Execute AND NOT fbCallMethod.Busy) THEN
			fbCallMethod.Execute := FALSE;
			IF (NOT fbCallMethod.Error) THEN
				eStateMethod := E_TrackClientState.ReleaseHandle;
			ELSE
				(* Error during get namespace index *)
				bErrorMethod := TRUE;
				nErrorMethodID := fbCallMethod.ErrorID;
				eStateMethod := E_TrackClientState.ReleaseHandle;
			END_IF
		ELSE
			fbCallMethod.Execute := TRUE;
		END_IF
	
	E_TrackClientState.ReleaseHandle:
		IF (fbReleaseHandleMethod.Execute AND NOT fbReleaseHandleMethod.Busy) THEN
			fbReleaseHandleMethod.Execute := FALSE;
			IF (bErrorMethod) THEN
				eStateMethod := E_TrackClientState.Error;	
				nHandleMethod := 0;
			ELSIF (NOT fbReleaseHandleMethod.Error) THEN
				nHandleMethod := 0;
				eStateMethod := E_TrackClientState.Connected;
			ELSE
				(* Error during release handle *)
				bErrorMethod := TRUE;
				nErrorMethodID := fbReleaseHandleMethod.ErrorID;
				nHandleMethod := 0;
				eStateMethod := E_TrackClientState.Disconnecting;
			END_IF
		ELSE
			fbReleaseHandleMethod.Execute := TRUE;
		END_IF
	
	E_TrackClientState.Disconnecting:
		bConnectedMethod := FALSE;
		IF (fbDisconnectMethod.Execute AND NOT fbDisconnectMethod.Busy) THEN
			fbDisconnectMethod.Execute := FALSE;
			IF (bErrorMethod) THEN
				eStateMethod := E_TrackClientState.Error;	
				nConnectHdlMethod := 0;				
			ELSIF (NOT fbDisconnectMethod.Error) THEN
				(* Disconnected *)
				nConnectHdlMethod := 0;
				eStateMethod := E_TrackClientState.Disconnected;
			ELSE
				(* Error during disconnection *)
				bErrorMethod := TRUE;
				nErrorMethodID := fbDisconnectMethod.ErrorID;
				nConnectHdlMethod := 0;
				eStateMethod := E_TrackClientState.Error;
			END_IF
		ELSE
			fbDisconnectMethod.Execute := TRUE;
		END_IF
	
	E_TrackClientState.Error:
		eStateMethod := E_TrackClientState.Disconnected;
		
END_CASE
END_METHOD

METHOD PROTECTED M_StateMachineNode_ADS : INT
VAR_INPUT
END_VAR
CASE eStateNode OF
	E_TrackClientState.Disconnected:
		bConnectedNode := FALSE;
		fbReadADS( bEnable := FALSE ); 
		IF (bEnable) THEN
			bErrorNode := FALSE;
			nErrorNodeID := 0;
			eStateNode := E_TrackClientState.Connected;
		END_IF
	
	E_TrackClientState.Connecting:
		eStateNode := E_TrackClientState.GetNamespaceIndex;
	
	E_TrackClientState.GetNamespaceIndex:
		eStateNode := E_TrackClientState.Connected;
	
	E_TrackClientState.Connected:	
//		bConnectedNode := TRUE;
		IF (NOT bEnable) THEN
			bConnectedNode := FALSE;
			eStateNode := E_TrackClientState.Disconnecting;
		ELSIF (M_InitNodeData_ADS()) THEN
			eStateNode := E_TrackClientState.Execute;			
		END_IF
		
	E_TrackClientState.GetHandle:
		eStateNode := E_TrackClientState.Execute;
	
	E_TrackClientState.Execute:
		fbReadADS(	bEnable:= TRUE, 
							eType:= E_ADS_Comm_Type.ADS_RD_FAST, 
							rInterval:= rReadInterval, 
							pLocalVar:= pReadNodeData, // M_InitNodeData_ADS 
							nLocalSize:= UDINT_TO_UINT(cbDataTotal), // M_InitNodeData_ADS
							sNetID:= sTrackServerNetID, 
							nPort:= nTrackServerPortNo, 
							sVarName:= sTrackServerSymbol, // M_InitNodeData_ADS
							bWriteError=> , 
							bReadError=> , 
							bParameterError=> );
		IF (fbReadADS.bReadError OR fbReadADS.bParameterError) THEN
			eStateNode := E_TrackClientState.Error;			
		ELSIF (fbReadADS.M_SendRecvCompleted()) THEN
			bConnectedNode := TRUE;
			fbReadADS( bEnable := FALSE );
			IF (bReadDecPointVehicleBusy) THEN
				// Reading of decision point vehicle data has completed! 
				bReadDecPointVehicleBusy := FALSE;
			
			ELSIF (eReadType = E_OPC_NodeType.Stations) THEN
				// Reading stations
				IF (F_StringCompNoCase(aReadStationData[iReadIndex].stStationData.sCellID, sCellID)) THEN
					// The read station belongs to this cell
					FOR iStatIndex := 1 TO 5 BY 1 DO
						 IF (aStations[iStatIndex].bPresent) THEN
							// Station is present, check station ID against the read station ID
							IF (F_StringCompNoCase(aReadStationData[iReadIndex].stStationData.sStationID, aStations[iStatIndex].sStationID)) THEN
								// Found matching station ID. Store it...
								iThisStationIndex[iStatIndex] := iReadIndex;
							END_IF
						ELSE
							iThisStationIndex[iStatIndex] := 0;
						END_IF
					END_FOR
				END_IF
			
			ELSIF (bReadDecPointCell) THEN
				// Reading cell data completed
				bReadDecPointCell := FALSE;
				bReadDecPointCellDone := TRUE;
			
			END_IF
			
			eStateNode := E_TrackClientState.Connected;
			iLastReadTimeMS := iReadTimeMS;
			iReadTimeMS := 0;
		END_IF
	
	E_TrackClientState.ReleaseHandle:
		eStateNode := E_TrackClientState.Connected;
	
	E_TrackClientState.Disconnecting:
		bConnectedNode := FALSE;
		eStateNode := E_TrackClientState.Disconnected;
	
	E_TrackClientState.Error:
		tonErrorReset.IN := TRUE;
		IF (tonErrorReset.Q) THEN
			tonErrorReset.IN := FALSE;
			eStateNode := E_TrackClientState.Disconnected;
		END_IF
		
END_CASE

// Read timer
iReadTimeMS := iReadTimeMS + 10;
END_METHOD

METHOD PROTECTED M_ThisCellDataIndex : UINT
VAR_INPUT
END_VAR
VAR
	i		: UINT;
END_VAR
// Locate the status data for this cell!

(*
// Check if a value is already found
IF (iThisCellIndex > 0) THEN 
	// Check previous found value
	IF (F_StringCompNoCase(	s1 := sCellID, s2 := aReadCellData[iThisCellIndex].stCell.sCellID)) THEN
		// Previous found value is OK
		;
	ELSE
		// Previous found value is NOT OK, find correct value
		iThisCellIndex := 0;
	END_IF
END_IF

IF (iThisCellIndex = 0) THEN 
	// Find correct value
	FOR i := 1 TO MM_MAX_NUMBER_OF_STATION_ELEMENTS BY 1 DO
		IF (F_StringCompNoCase(sCellID, s2 := aReadCellData[i].stCell.sCellID)) THEN
			// Correct cell ID found
			iThisCellIndex := i;
			EXIT;
		END_IF
	END_FOR
END_IF
*)

M_ThisCellDataIndex := iThisCellIndex;
END_METHOD

METHOD PROTECTED M_UpdateStatus : BOOL
VAR_INPUT
END_VAR
VAR
	iBuffer				: UINT;
	iVehicleID			: UINT;
	iVehicleIndex		: UINT;
	bDataChanged		: BOOL;
END_VAR
// Update status values

// Check if LC allows to change status data
IF (stAdditionalDataIn.MESHandShakes.DataChangeStatusTransportStatus = stStatus.DataChange) THEN
	////////////////////////////////////////////////////////////////////////////////////////////////////////////////////////////////////
	// Vehicles
	////////////////////////////////////////////////////////////////////////////////////////////////////////////////////////////////////
	iVehicleIndex := 1;
	iVehicleID := 1;
	bDataChanged := FALSE;
	MEMSET(ADR(stStatus.Carrier), 0, SIZEOF(stStatus.Carrier));
	WHILE iVehicleID < MM_MAX_NUMBER_OF_VEHICLE_ELEMENTS DO
	
		IF ((aReadVehicleData[iVehicleID].stVehicle.nVehicleID > 0) AND
			(aReadVehicleData[iVehicleID].stVehicle.bDataValid) ) THEN
			// Vehicle has valid data
			IF ((aReadVehicleData[iVehicleID].stVehicle.sOwnerCell = sCellID) AND M_CheckVehicleOwned(aReadVehicleData[iVehicleID].stVehicle.nVehicleID)) THEN
				// Vehicle belongs to this cell
				stStatus.Carrier[iVehicleIndex].CarrierID := aReadVehicleData[iVehicleID].stVehicle.sCarrierID;
				stStatus.Carrier[iVehicleIndex].CarriersInPackage := aReadVehicleData[iVehicleID].stVehicle.nTicketSize; 
				stStatus.Carrier[iVehicleIndex].CarrierStatus := aReadVehicleData[iVehicleID].stVehicle.nState;
				stStatus.Carrier[iVehicleIndex].CurrentPath := aReadVehicleData[iVehicleID].stVehicle.nPathID;
				stStatus.Carrier[iVehicleIndex].CurrentPosition := aReadVehicleData[iVehicleID].stVehicle.fPosition;
				stStatus.Carrier[iVehicleIndex].CurrentStation := aReadVehicleData[iVehicleID].stVehicle.sCurrentStationID;
				stStatus.Carrier[iVehicleIndex].JobID := aReadVehicleData[iVehicleID].stVehicle.sJobID;
				IF (aReadVehicleData[iVehicleID].stVehicle.sLastScan <> '') THEN
					stStatus.Carrier[iVehicleIndex].LastScan := STRING_TO_DT(CONCAT('DT#', aReadVehicleData[iVehicleID].stVehicle.sLastScan));
				END_IF
				stStatus.Carrier[iVehicleIndex].Material := aReadVehicleData[iVehicleID].stVehicle.bMaterial;
				stStatus.Carrier[iVehicleIndex].MaterialID := aReadVehicleData[iVehicleID].stVehicle.sMaterialID;
				stStatus.Carrier[iVehicleIndex].Priority := aReadVehicleData[iVehicleID].stVehicle.nPriority;
				IF (aReadVehicleData[iVehicleID].stVehicle.sTargetStationID <> '') THEN
					stStatus.Carrier[iVehicleIndex].TargetReached := (aReadVehicleData[iVehicleID].stVehicle.sTargetStationID = aReadVehicleData[iVehicleID].stVehicle.sCurrentStationID);
				ELSE
					stStatus.Carrier[iVehicleIndex].TargetReached := FALSE;
				END_IF
				// Update Target Reached Counter
				IF ((aOldVehicleData[iVehicleID].sCurrentStationID = '') AND (aReadVehicleData[iVehicleID].stVehicle.sCurrentStationID <> '')) THEN
					IF (aReadVehicleData[iVehicleID].stVehicle.sTargetStationID = aReadVehicleData[iVehicleID].stVehicle.sCurrentStationID) THEN
						// First scan this vehicle is on position
						aOldVehicleTargetReachedCnt[iVehicleID] := aOldVehicleTargetReachedCnt[iVehicleID] + 1;
						IF (aOldVehicleTargetReachedCnt[iVehicleID] >= 100) THEN
							aOldVehicleTargetReachedCnt[iVehicleID] := 0;
						END_IF
					END_IF
				END_IF
				stStatus.Carrier[iVehicleIndex].TargetReachedCounter := (iThisCellIndex * 100) + aOldVehicleTargetReachedCnt[iVehicleID];
				stStatus.Carrier[iVehicleIndex].TargetStation := aReadVehicleData[iVehicleID].stVehicle.sTargetStationID;
				stStatus.Carrier[iVehicleIndex].Ticket := aReadVehicleData[iVehicleID].stVehicle.nTicket;
				stStatus.Carrier[iVehicleIndex].Tool := aReadVehicleData[iVehicleID].stVehicle.bTool;
				stStatus.Carrier[iVehicleIndex].ToolID := aReadVehicleData[iVehicleID].stVehicle.sToolID;
				stStatus.Carrier[iVehicleIndex].ValidData := aReadVehicleData[iVehicleID].stVehicle.bDataValid;
				stStatus.Carrier[iVehicleIndex].NOK := aReadVehicleData[iVehicleID].stVehicle.bNOK;
				
				iVehicleIndex := iVehicleIndex + 1;
				
				// Compare with old vehicle data
				bDataChanged := bDataChanged OR M_UpdateStatusCompare(iVehicleID);
			END_IF
		END_IF
	
		// Save as old vehicle data
		aOldVehicleData[iVehicleID] := aReadVehicleData[iVehicleID].stVehicle;
		
		// Next vehicle
		iVehicleID := iVehicleID + 1;
	END_WHILE
	stStatus.NumberOfCarriers := (iVehicleIndex - 1);
	// Check if number of carriers has changed and update data if it has
	IF (stStatus.NumberOfCarriers <> iOldVehicleCount) THEN
		bDataChanged := TRUE;
		iOldVehicleCount := stStatus.NumberOfCarriers;
	END_IF
	
	// Check if data has changed
	IF (bDataChanged OR bForceVehicleUpdateOPC) THEN
		bForceVehicleUpdateOPC := FALSE;
		stStatus.DataChange := stStatus.DataChange + 1;
	END_IF
	
	
	////////////////////////////////////////////////////////////////////////////////////////////////////////////////////////////////////
	// Stations
	////////////////////////////////////////////////////////////////////////////////////////////////////////////////////////////////////
	iStation := iStation + 1;
	IF (iStation > 5) THEN
		iStation := 1;
	END_IF
	// Station ID
	stStatus.StationBuffer[iStation].StationID := aStations[iStation].sStationID;
	IF (aStations[iStation].bPresent) THEN
		// Station 1 (input) values (placed at the first Pre-buffer index!)
		stStatus.StationBuffer[iStation].PreBuffer.BufferIndex[1].Present := aStations[iStation].stStationData1.bPresent;
		stStatus.StationBuffer[iStation].PreBuffer.BufferIndex[1].CarrierID := M_VehicleIDToCarrierID(aStations[iStation].stStationData1.nCurrentVehicleID);
		stStatus.StationBuffer[iStation].PreBuffer.BufferIndex[1].Ticket := aStations[iStation].stStationData1.nTicket;
		// Station 2 (output) values (placed at the first Post-buffer index!)
		stStatus.StationBuffer[iStation].PostBuffer.BufferIndex[1].Present := aStations[iStation].stStationData2.bPresent;
		stStatus.StationBuffer[iStation].PostBuffer.BufferIndex[1].CarrierID := M_VehicleIDToCarrierID(aStations[iStation].stStationData2.nCurrentVehicleID);
		stStatus.StationBuffer[iStation].PostBuffer.BufferIndex[1].Ticket := aStations[iStation].stStationData2.nTicket;
		// Buffers
		stStatus.StationBuffer[iStation].PreBuffer.Capacity := 0;
		stStatus.StationBuffer[iStation].PreBuffer.CapacityUsed := 0;
		stStatus.StationBuffer[iStation].PostBuffer.Capacity := 0;
		stStatus.StationBuffer[iStation].PostBuffer.CapacityUsed := 0;
		FOR iBuffer := 1 TO MM_MAX_BUFFER_INDEX BY 1 DO
			// Pre-buffer capacity
			IF (aStations[iStation].astPreBuffer[iBuffer].bPresent) THEN
				stStatus.StationBuffer[iStation].PreBuffer.Capacity := stStatus.StationBuffer[iStation].PreBuffer.Capacity + 1;
			END_IF
			// Pre-buffer used capacity
			IF (aStations[iStation].astPreBuffer[iBuffer].nCurrentVehicleID > 0) THEN
				stStatus.StationBuffer[iStation].PreBuffer.CapacityUsed := stStatus.StationBuffer[iStation].PreBuffer.CapacityUsed + 1;
			END_IF
			// Pre-buffer values
			stStatus.StationBuffer[iStation].PreBuffer.BufferIndex[iBuffer+1].Present := aStations[iStation].astPreBuffer[iBuffer].bPresent;
			stStatus.StationBuffer[iStation].PreBuffer.BufferIndex[iBuffer+1].CarrierID := M_VehicleIDToCarrierID(aStations[iStation].astPreBuffer[iBuffer].nCurrentVehicleID);
			stStatus.StationBuffer[iStation].PreBuffer.BufferIndex[iBuffer+1].Ticket := aStations[iStation].astPreBuffer[iBuffer].nTicket;
			// Post-buffer capacity
			IF (aStations[iStation].astPostBuffer[iBuffer].bPresent) THEN
				stStatus.StationBuffer[iStation].PostBuffer.Capacity := stStatus.StationBuffer[iStation].PostBuffer.Capacity + 1;
			END_IF
			// Post-buffer used capacity
			IF (aStations[iStation].astPostBuffer[iBuffer].nCurrentVehicleID > 0) THEN
				stStatus.StationBuffer[iStation].PostBuffer.CapacityUsed := stStatus.StationBuffer[iStation].PostBuffer.CapacityUsed + 1;
			END_IF
			// Post-buffer values
			stStatus.StationBuffer[iStation].PostBuffer.BufferIndex[iBuffer+1].Present := aStations[iStation].astPostBuffer[iBuffer].bPresent;
			stStatus.StationBuffer[iStation].PostBuffer.BufferIndex[iBuffer+1].CarrierID := M_VehicleIDToCarrierID(aStations[iStation].astPostBuffer[iBuffer].nCurrentVehicleID);
			stStatus.StationBuffer[iStation].PostBuffer.BufferIndex[iBuffer+1].Ticket := aStations[iStation].astPostBuffer[iBuffer].nTicket;
			
		END_FOR
	END_IF

END_IF
END_METHOD

/// Compares two vehicle data sets. Returns TRUE if different
METHOD PROTECTED M_UpdateStatusCompare : BOOL
VAR_INPUT
	iVehicleID		: UINT;
END_VAR

// Check for changes (uncomment/comment to choose which values should be compared!)
IF ( (iVehicleID >= 1) AND (iVehicleID <= MM_MAX_NUMBER_OF_VEHICLE_ELEMENTS) ) THEN
	IF ( 	(aReadVehicleData[iVehicleID].stVehicle.bDataValid <> aOldVehicleData[iVehicleID].bDataValid) OR
			(aReadVehicleData[iVehicleID].stVehicle.bMaterial <> aOldVehicleData[iVehicleID].bMaterial) OR
			(aReadVehicleData[iVehicleID].stVehicle.bNOK <> aOldVehicleData[iVehicleID].bNOK) OR
			(aReadVehicleData[iVehicleID].stVehicle.bTool <> aOldVehicleData[iVehicleID].bTool) OR
			(aReadVehicleData[iVehicleID].stVehicle.bVehiclePresent <> aOldVehicleData[iVehicleID].bVehiclePresent) OR
//			(aReadVehicleData[iVehicleID].stVehicle.fPosition <> aOldVehicleData[iVehicleID].fPosition) OR
//			(aReadVehicleData[iVehicleID].stVehicle.fTargetPosition <> aOldVehicleData[iVehicleID].fTargetPosition) OR
//			(aReadVehicleData[iVehicleID].stVehicle.fVelocity <> aOldVehicleData[iVehicleID].fVelocity) OR
//			(aReadVehicleData[iVehicleID].stVehicle.nPathID <> aOldVehicleData[iVehicleID].nPathID) OR
			(aReadVehicleData[iVehicleID].stVehicle.nPriority <> aOldVehicleData[iVehicleID].nPriority) OR
//			(aReadVehicleData[iVehicleID].stVehicle.nState <> aOldVehicleData[iVehicleID].nState) OR
//			(aReadVehicleData[iVehicleID].stVehicle.nTargetPathID <> aOldVehicleData[iVehicleID].nTargetPathID) OR
			(aReadVehicleData[iVehicleID].stVehicle.nTicket <> aOldVehicleData[iVehicleID].nTicket) OR
			(aReadVehicleData[iVehicleID].stVehicle.nTicketSize <> aOldVehicleData[iVehicleID].nTicketSize) OR
			(aReadVehicleData[iVehicleID].stVehicle.nVehicleID <> aOldVehicleData[iVehicleID].nVehicleID) OR
			(aReadVehicleData[iVehicleID].stVehicle.sCarrierID <> aOldVehicleData[iVehicleID].sCarrierID) OR
			(aReadVehicleData[iVehicleID].stVehicle.sCurrentStationID <> aOldVehicleData[iVehicleID].sCurrentStationID) OR
			(aReadVehicleData[iVehicleID].stVehicle.sJobID <> aOldVehicleData[iVehicleID].sJobID) OR
			(aReadVehicleData[iVehicleID].stVehicle.sLastScan <> aOldVehicleData[iVehicleID].sLastScan) OR
			(aReadVehicleData[iVehicleID].stVehicle.sMaterialID <> aOldVehicleData[iVehicleID].sMaterialID) OR
			(aReadVehicleData[iVehicleID].stVehicle.sOwnerCell <> aOldVehicleData[iVehicleID].sOwnerCell) OR
			(aReadVehicleData[iVehicleID].stVehicle.sTargetStationID <> aOldVehicleData[iVehicleID].sTargetStationID) OR
			(aReadVehicleData[iVehicleID].stVehicle.sToolID <> aOldVehicleData[iVehicleID].sToolID)
		) THEN
		// Change detected. Return TRUE
		M_UpdateStatusCompare := TRUE;
		RETURN;
	END_IF
END_IF

M_UpdateStatusCompare := FALSE;
END_METHOD

METHOD PROTECTED M_VehicleIDToCarrierID : STRING(30)
VAR_INPUT
	nVehicleID		: UINT;
END_VAR

VAR
	i: INT;
END_VAR


IF (nVehicleID > 0 AND nVehicleID <= MM_MAX_NUMBER_OF_VEHICLE_ELEMENTS) THEN
	M_VehicleIDToCarrierID := aReadVehicleData[nVehicleID].stVehicle.sCarrierID;
	
ELSE
	M_VehicleIDToCarrierID := '';
	
END_IF
END_METHOD

/// Adds a vehicle to list of vehicles to read evnet-driven data from
METHOD M_VehicleToReadAdd : BOOL
VAR_INPUT
	iVehicleNo		: UINT;
END_VAR
VAR
	i				: UINT;
END_VAR

IF (iVehicleNo > 0 AND iVehicleNo <= MM_MAX_NUMBER_OF_VEHICLE_ELEMENTS) THEN
	FOR i := 1 TO MM_MAX_NUMBER_OF_VEHICLE_ELEMENTS BY 1 DO
		IF (anVehiclesToRead[i] = iVehicleNo) THEN
			// Vehicle is already added
			M_VehicleToReadAdd := TRUE;
			RETURN;
		
		ELSIF (anVehiclesToRead[i] = 0) THEN
			// Empty index found
			anVehiclesToRead[i] := iVehicleNo;
			M_VehicleToReadAdd := TRUE;
			RETURN;
			
		END_IF
	END_FOR
	
ELSE
	// Not within range
	M_VehicleToReadAdd := FALSE;
	
END_IF
END_METHOD

/// Removes a vehicle from list of vehicles to read evnet-driven data from
METHOD M_VehicleToReadRemove : BOOL
VAR_INPUT
	iVehicleNo		: UINT;
END_VAR
VAR
	i				: UINT;
END_VAR

IF (iVehicleNo > 0 AND iVehicleNo <= MM_MAX_NUMBER_OF_VEHICLE_ELEMENTS) THEN
	FOR i := 1 TO MM_MAX_NUMBER_OF_VEHICLE_ELEMENTS BY 1 DO
		IF (anVehiclesToRead[i] = iVehicleNo) THEN
			// Vehicle is found
			anVehiclesToRead[i] := 0;
			M_VehicleToReadRemove := TRUE;
			RETURN;
			
		END_IF
	END_FOR
	
ELSE
	// Not within range
	M_VehicleToReadRemove := FALSE;
	
END_IF
END_METHOD

PROPERTY PUBLIC P_bForceVehicleUpdateOPC : BOOL
GET
P_bForceVehicleUpdateOPC := bForceVehicleUpdateOPC;
END_GET
SET
bForceVehicleUpdateOPC := P_bForceVehicleUpdateOPC;
END_SET
END_PROPERTY

/// When TRUE it is OK to run DecisionPoint, ExitPoint and Buffer handling
PROPERTY PUBLIC P_bTrackReady : BOOL
GET
// TRUE if track client is ready to use
P_bTrackReady := bEnable AND bConnectedMethod AND bConnectedNode AND bTrackInitDone AND (eTrackState = E_TrackState.Started);
END_GET
END_PROPERTY

PROPERTY PUBLIC P_eCellType : E_CellType
GET
P_eCellType := eCellType;
END_GET
SET
eCellType := P_eCellType;
END_SET
END_PROPERTY

PROPERTY PUBLIC P_nTrackserverPort : UINT
GET
P_nTrackserverPort := nTrackServerPortNo;
END_GET
SET
nTrackServerPortNo := P_nTrackserverPort;
END_SET
END_PROPERTY

PROPERTY PUBLIC P_rErrorResetDelay : REAL
GET
P_rErrorResetDelay := rErrorResetDelay;
END_GET
SET
rErrorResetDelay := P_rErrorResetDelay;
END_SET
END_PROPERTY

PROPERTY PUBLIC P_rPollingInterval : REAL
GET
P_rPollingInterval := rReadInterval;
END_GET
SET
rReadInterval := P_rPollingInterval;
END_SET
END_PROPERTY

PROPERTY PUBLIC P_sCellID : STRING(30)
GET
P_sCellID := sCellID;
END_GET
SET
sCellID := F_ToUCase(P_sCellID);
END_SET
END_PROPERTY

PROPERTY PUBLIC P_sNextStationOnTrack : STRING(30)
GET
P_sNextStationOnTrack := sNextStationOnTrack;
END_GET
SET

IF (LEN(P_sNextStationOnTrack) > 0) THEN
	sNextStationOnTrack := P_sNextStationOnTrack;
END_IF
END_SET
END_PROPERTY

PROPERTY PUBLIC P_sTrackserverNetID : STRING
GET
P_sTrackserverNetID := sTrackServerNetID;
END_GET
SET
sTrackServerNetID := P_sTrackserverNetID;
END_SET
END_PROPERTY

PROPERTY PUBLIC P_sTrackserverURL : STRING
GET
P_sTrackserverURL := sTrackServerUrl;
END_GET
SET
sTrackServerUrl := P_sTrackserverURL;
END_SET
END_PROPERTY

END_FUNCTION_BLOCK

(* stored: Version 1.1.0.1, ProductVersion 3.1.4024.5
   POU FB_TrackClient_Basic: Id {1ac5e215-eb59-4502-99b0-c2a46163e22f}, SpecialFunc None
   Method M_CallAddPath: Id {e402ea3c-7941-4e8e-9950-0a0e536fd4bc}
   Method M_CallAddPathSegment: Id {b299dbc9-6201-4492-afc6-2d3445661ab5}
   Method M_CallAddReservation: Id {8463457c-3357-4365-b2ca-16e3af92ba18}
   Method M_CallAddStationDouble: Id {4ac951a4-17d3-4c18-8138-422b88041efa}
   Method M_CallAddStationSingle: Id {c2075884-4710-46d6-b9e2-6200882a642f}
   Method M_CallAddTrafficLight: Id {54cb9d7a-29b8-49d8-b018-b9c14e7e7a57}
   Method M_CallAdjustBufferPosition: Id {d74a7a82-68ca-4e44-870e-9ccc8dfe228c}
   Method M_CallEnableStation: Id {2df14879-a9d2-4c81-a5b8-7b562f03d8cc}
   Method M_CallGetCellIndex: Id {a6243e62-ba37-4885-95a6-6c7f3c673478}
   Method M_CallGetPathSegmentVehicleCount: Id {d2d1be27-cbbe-4456-ac72-3b33b1e14a78}
   Method M_CallMoveVehicleStatus: Id {14afa176-ece5-4d45-9676-2b8f4c0291b6}
   Method M_CallMoveVehicleToBuffer: Id {d022b077-1f98-41a3-8d09-690839470c28}
   Method M_CallMoveVehicleToDecisionPoint: Id {229ffaa2-54ab-46e5-8cee-d6eabeed20d3}
   Method M_CallMoveVehicleToPosition: Id {25ee421d-a63f-44f1-b077-113ad1b8812b}
   Method M_CallMoveVehicleToScanner: Id {200c491c-0472-4a16-a7f2-753209075ebf}
   Method M_CallMoveVehicleToStationIn: Id {99b48e28-5891-493a-afd0-9ec1883273c5}
   Method M_CallMoveVehicleToStationOut: Id {4f44d3ad-713f-4108-8557-f96306db0c2d}
   Method M_CallRemovePath: Id {92a6b858-3c08-4dea-ae3b-f5ef1c1f7bcb}
   Method M_CallRemovePathSegment: Id {89ef444e-206c-4289-83a8-303e94a443c2}
   Method M_CallRemoveReservation: Id {445ba283-972e-489b-9fd4-6609fe655ab5}
   Method M_CallRemoveStation: Id {e256acd0-5eb0-46bc-9fb2-66a0bbff7d33}
   Method M_CallRemoveTrafficLight: Id {5c7df096-ff73-4ea2-bbd4-0977b8085d14}
   Method M_CallResetPath: Id {d14bbf22-85cb-4a04-854c-25a775e0ea3e}
   Method M_CallResumePath: Id {dd3456c4-41fd-46f5-9378-e1fd4dd8cab0}
   Method M_CallSetTrafficLightColor: Id {39a7e5e7-dcf3-4537-b684-fca830d15aa8}
   Method M_CallStartPath: Id {8a8a0f75-2db0-41da-b49f-94dd573e7154}
   Method M_CallSuspendPath: Id {557446d8-92e3-41af-abfa-2649e650b0cc}
   Method M_CallTrafficLightColor: Id {f77855b9-801c-43b0-aba4-3a7c320e868e}
   Method M_CallUpdateStationBuffer: Id {c5e96520-9256-4b65-9f9c-03d2b61e42bb}
   Method M_CallUpdateVehicleMappingData: Id {58eb1d4d-9766-4816-bba9-5e7797d1d67f}
   Method M_CallUpdateVehicleMontage: Id {b034f17a-5d35-4c96-9dbf-a079f59588be}
   Method M_CallUpdateVehicleOwner: Id {5b44b485-93bc-45c9-8b6a-282eaee4e001}
   Method M_CallUpdateVehicleReservationData: Id {4b57a1ab-f899-4caf-ae31-65d088b92f63}
   Method M_CallUpdateVehicleReworkData: Id {35e08d3d-3091-4034-b597-597ed59aaf02}
   Method M_CarrierIDToVehicleID: Id {08a565de-8270-4e6c-be7d-d28b35e5c0e0}
   Method M_CheckStationIndex: Id {17b0b2e4-1e13-461c-9a9f-fc544d74087a}
   Method M_CheckStationsRead: Id {c0200038-6928-4202-b86b-98923d328126}
   Method M_CheckVehicleEventRead: Id {afde6db3-8165-4ca2-bc1e-cfee91df1de6}
   Method M_CheckVehicleOwned: Id {e41741fc-4227-442f-b07b-3e2869eddce6}
   Method M_CheckVehicleSurvail: Id {57a1d781-5991-4c44-834a-d4fcef59c758}
   Method M_ClearAll: Id {39d6c25d-bfba-40b0-9d86-85672d6eb51a}
   Method M_CommandData: Id {904b5ce0-46cc-4181-91bc-a3e47c4bbb8c}
   Method M_CopyAndClearBufferData: Id {be8b5ba0-b2c5-4458-931a-caaad8c7d2d1}
   Method M_CopyBufferData: Id {d04f8618-5494-4b8a-a309-80314dd3e340}
   Method M_DefinePath: Id {d6dd8c8b-6c7e-4e6e-a2ed-ce346467b26a}
   Method M_DefinePathSegment: Id {ef3e9644-bd4c-4eb5-b126-cc812d729970}
   Method M_DefineStation: Id {9ef508f7-a4c4-48b8-8a54-b8a3b8faf0f2}
   Method M_DefineStationBufferAdjust: Id {ea76cb0a-33c6-400e-83de-2b7df949d5d7}
   Method M_DefineTrafficLight: Id {e9787981-10aa-43a3-953d-e2259c325ef5}
   Method M_EnableStation: Id {9438130a-40b8-466a-b73c-7eeb3aec0a92}
   Method M_ErrorWarning: Id {06aa7e66-21cb-4c9d-b9a5-322fe9803221}
   Method M_ErrorWarningObj: Id {97ecedeb-8310-4597-8db4-64c05fc8f0bf}
   Method M_ExtraVehicleAdd: Id {52fed8e5-609f-420b-b891-df588ae939ad}
   Method M_ExtraVehicleRemove: Id {488ac611-b893-4238-ba10-e6edae0f29b1}
   Method M_Init: Id {1750c38c-e1c3-435a-a405-b6117cd09d25}
   Method M_InitMethodData: Id {19ca9e8b-89b7-47f8-a1cd-d258530813a4}
   Method M_InitNodeData: Id {2ec3e5fa-b79a-4527-9486-48de86728ba0}
   Method M_InitNodeData_ADS: Id {5984c523-b795-4b39-9e4a-723ce44ca072}
   Method M_InitNodeData_OPCUA: Id {d0af0184-d04d-4703-a126-3478d4c3c72f}
   Method M_MappingData: Id {556fccca-69db-43f4-b7b4-ab5b0d065e23}
   Method M_ReworkData: Id {fb0c97a7-e083-4c09-9fc7-0083f6bba4ec}
   Method M_Run: Id {32f5619d-9c61-45ef-983b-857f7d3984c4}
   Method M_StateMachine: Id {75832c14-cca9-41ab-90e4-a04ce178e3d7}
   Method M_StateMachineMethod: Id {d89a46e6-0e6c-475c-b1d1-e8c3887e2e35}
   Method M_StateMachineNode_ADS: Id {6dcba053-df50-46f8-98a7-c28bc41e7c44}
   Method M_ThisCellDataIndex: Id {11157ab8-8c73-4a36-913e-bbb5350ce1c2}
   Method M_UpdateStatus: Id {5f0f8b17-844e-4675-bc4e-f1b959826218}
   Method M_UpdateStatusCompare: Id {7d09dc7d-0580-4962-897a-5c7e9c84fa80}
   Method M_VehicleIDToCarrierID: Id {1010ebd7-d6ed-40d5-97a1-367a1bc6d91f}
   Method M_VehicleToReadAdd: Id {a0aa4f66-4471-4cda-a80e-bc2f02e6f23c}
   Method M_VehicleToReadRemove: Id {5f83c716-b2a2-4298-a7b9-54128794aacb}
   Property P_bForceVehicleUpdateOPC: Id {e3de05d9-bf15-4006-8645-6bca37fa13a2}
   Get Get: Id {890e6faa-0b13-4388-985b-1f92d2037962}
   Set Set: Id {f73b0f77-ee39-49f4-bcfd-a3070f03a59d}
   Property P_bTrackReady: Id {563c5a2a-b947-4cfc-b8ff-ede349f496cc}
   Get Get: Id {4d1cb31f-2455-4823-9437-6f43cbe07729}
   Property P_eCellType: Id {f8b89a3c-d4eb-4974-a116-e6eec1810f83}
   Get Get: Id {006cbb3d-a5c5-4ee1-9b95-11aef70b137a}
   Set Set: Id {14cc0dd7-2e32-465b-a1bc-9e64e02fe4e8}
   Property P_nTrackserverPort: Id {9ee8c101-fd90-4b09-85be-1e0628572d3d}
   Get Get: Id {0914898f-abcb-4ecd-8f3c-551f5fea0a19}
   Set Set: Id {3e945c77-02b4-4deb-8672-0c5c041f42b7}
   Property P_rErrorResetDelay: Id {3d49e448-b86b-4ee0-8ddb-1b333b59596c}
   Get Get: Id {72d8357e-1e35-4de1-abef-6ad5331a419a}
   Set Set: Id {b972263f-3cd7-4b94-9d48-32641e5a40f7}
   Property P_rPollingInterval: Id {f49f6fd9-e679-404d-8a03-5145bc48e193}
   Get Get: Id {28d08fd3-eed1-4ca6-a523-f1fdc1b8ae50}
   Set Set: Id {ed2c62b3-522f-4f15-9696-e47959a2fb8d}
   Property P_sCellID: Id {e88ab857-2756-4b4a-8845-c2333efc8a0b}
   Get Get: Id {6d189475-286d-4e02-8d7a-6352c6277a07}
   Set Set: Id {8187e086-961e-4f87-8540-0fdf96eb0619}
   Property P_sNextStationOnTrack: Id {b803813b-9aaf-4e85-82f8-218f9f9b1347}
   Get Get: Id {12d2266c-e012-4698-84b4-8ba60a400ef2}
   Set Set: Id {9a26e180-bf0c-4868-8917-397b31d1616f}
   Property P_sTrackserverNetID: Id {f4ab271d-2693-4e10-9d44-fa9a4099a6c8}
   Get Get: Id {038c7f3c-fba8-4975-a833-56cbc64fb8f0}
   Set Set: Id {616ebaec-77fa-4482-87ee-b39f2ebc9057}
   Property P_sTrackserverURL: Id {92aa76bc-cc3a-456f-bc80-2077a04fc128}
   Get Get: Id {b9d513db-0ae6-416a-9357-745bcd76d8f2}
   Set Set: Id {23a8a54b-09bc-4372-9f66-a6a892aaabb1} *)
